# EPICS substitutions: synApps_6_1/support/motor-R7-1/modules/motorFaulhaber/iocs/faulhaberIOC/iocBoot/iocFaulhaber/MCDC2805.substitutions
file "$(MOTOR)/db/motor.db"
{
pattern
{P,          N,     M,     DTYP,         C, S, DESC,          EGU,    DIR,	VELO, VBAS, ACCL, BDST, BVEL, BACC, MRES, PREC, DHLM, DLLM, INIT}
{faulhaber:, 1, "m$(N)", "MCDC2805",     0, 0, "motor $(N)", degrees, Pos, 10,    0.,   1.,   0,    1,    .2,   1e-3, 3,    100,  -100, ""}
}
